(* CODESYS project 4.project

Project tree, tasks and I/O mapping:
  Device : CODESYS Control Win V3, 3S - Smart Software Solutions GmbH, order no. 305021, version 3.5.11.30
    application Application
      libraries: Standard, * (System)
      task MainTask (cyclic, interval t#20ms, priority 1) calls PLC_PRG
      program PLC_PRG [LD]
*)

// Device/Application/PLC_PRG
PROGRAM PLC_PRG
VAR
	S1: BOOL; //SENSOR DA MESA DO OPERADOR
	KM1: BOOL; //M1 IDA
	KM0: BOOL; //M1 VOLTA
	// FIM DE CURSO 1
	FC1: BOOL;
	KM2: BOOL;
	// TEMPORISADOR DO M2
	TON_0: TON;
	// FIM DE CURSO 2 - MOTOR 3
	FC2: BOOL;
	KM3: BOOL;
	TON_1: TON;
END_VAR

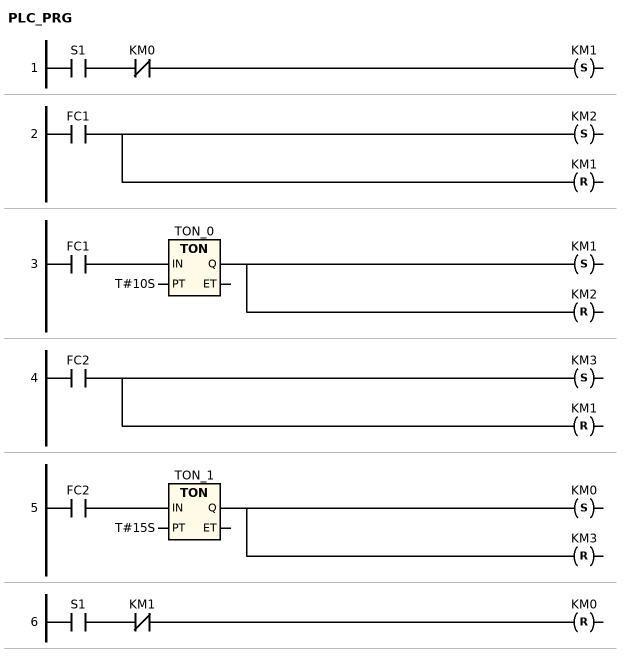
// NETWORK 1
KM1 S= S1 AND NOT KM0;

// NETWORK 2
KM2 S= FC1;
KM1 R= FC1;

// NETWORK 3
TON_0(IN := FC1, PT := T#10S); // TON
KM1 S= TON_0.Q;
KM2 R= TON_0.Q;

// NETWORK 4
KM3 S= FC2;
KM1 R= FC2;

// NETWORK 5
TON_1(IN := FC2, PT := T#15S); // TON
KM0 S= TON_1.Q;
KM3 R= TON_1.Q;

// NETWORK 6
KM0 R= S1 AND NOT KM1;

END_PROGRAM
